KUKA KRL program: ab_st_60301.src, ab_st_60301.dat

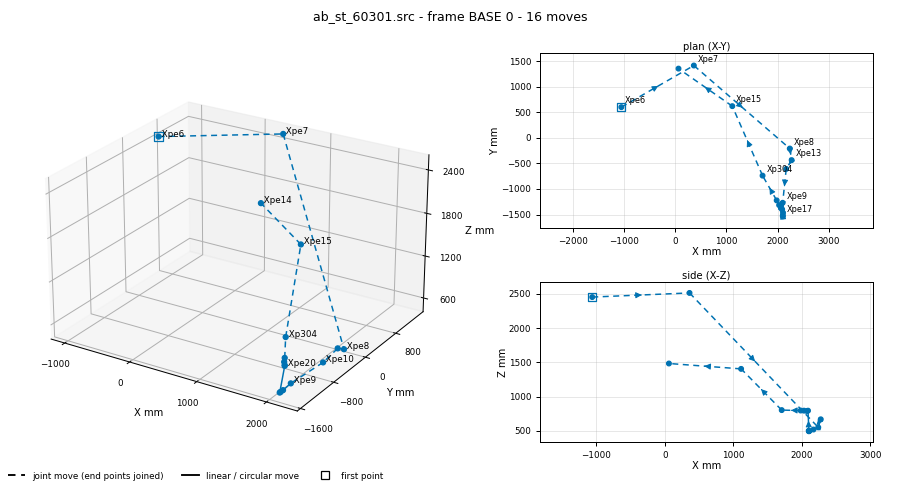
[picture p0: tool path of ab_st_60301.src in frame BASE 0, 16 of 16 moves have a stored position in this frame; points joined in program order, loops and branches not executed]
--- ab_st_60301.src ---
&ACCESS RV2
&REL 437
&COMMENT Deposita Frontal na Geo
&PARAM TEMPLATE = C:\KRC\Roboter\Template\vorgabe
&PARAM EDITMASK = *
DEF ab_st_60301( )
;FOLD INI;%{PE}%V3.2.0,%MKUKATPBASIS,%CINIT,%VCOMMON,%P
;FOLD BAS INI;%{E}%V3.2.0,%MKUKATPBASIS,%CINIT,%VINIT,%P
GLOBAL INTERRUPT DECL 3 WHEN $STOPMESS==TRUE DO IR_STOPM ( )
INTERRUPT ON 3
BAS (#INITMOV,0 )
;ENDFOLD (BAS INI)
;FOLD A20 INI;%{E}%V3.2.0,%MKUKATPA20,%CINIT,%VINIT,%P
IF ARC20==TRUE THEN
A20 (ARC_INI)
INTERRUPT DECL 6 WHEN $CYCFLAG[3]==FALSE DO A20(TECH_STOP2)
ENDIF
;ENDFOLD (A20 INI)
;FOLD A10 INI;%{E}%V3.2.0,%MKUKATPARC,%CINIT,%VINIT,%P
IF A10_OPTION==#ACTIVE THEN
INTERRUPT DECL 4 WHEN $CYCFLAG[2]==FALSE DO A10 (#APPL_ERROR)
INTERRUPT DECL 7 WHEN A_ARC_SWI==#ACTIVE DO A10 (#ARC_SEAM)
INTERRUPT DECL 5 WHEN A_FLY_ARC==TRUE DO A10 (#HPU_ARC)
INTERRUPT  ON 5
A10_INI ( )
ENDIF
;ENDFOLD (A10 INI)
;FOLD GRIPPER INI;%{E}%V3.2.0,%MKUKATPGRIPPER,%CINIT,%VINIT,%P
USER_GRP(0,DUMMY,DUMMY,GDEFAULT)
;ENDFOLD (GRIPPER INI)
;FOLD SPOT INI;%{E}%V3.2.0,%MKUKATPSPOT,%CINIT,%VINIT,%P
USERSPOT(#INIT)
;ENDFOLD (SPOT INI)
;FOLD TOUCHSENSE INI;%{E}%V3.2.0,%MKUKATPTS,%CINIT,%VINIT,%P
IF H70_OPTION THEN
INTERRUPT DECL 15 WHEN $MEAS_PULSE[TOUCH_I[TOUCH_ACTIVE].IN_NR] DO H70 (6,CD0 )
INTERRUPT DECL 16 WHEN $ZERO_MOVE DO H70 (7,CD0 )
INTERRUPT DECL 17 WHEN $TECHPAR_C[FG_TOUCH,8]>0.5 DO H70 (8,CD0)
H70 (1,CD0 )
ENDIF
;ENDFOLD (TOUCHSENSE INI)
;FOLD USER INI;%{E}%V3.2.0,%MKUKATPUSER,%CINIT,%VINIT,%P
;Make your modifications here
;ENDFOLD (USER INI)
;ENDFOLD (INI)

; Caracterização dos meios de produção:
; Versão Atual:
; 19/07/2013 12:00 Name: P13.060-R3 CHANGES: Deposita Frontal Accelo
; na Geobox

chk_w3_wechs_ok ( )        ; ERIFICAÇÃO DE FERRAMENTA: GRIPPER

;FOLD PTP pe6  Vel= 100 % PDAT62 Tool[3]:Gripper Frontal Accelo Base[0];%{PE}%R 4.1.16,%MKUKATPBASIS,%CMOVE,%VPTP,%P 1:PTP, 2:pe6, 3:, 5:100, 7:PDAT62
$BWDSTART = FALSE
PDAT_ACT=PPDAT62
BAS(#PTP_DAT)
FDAT_ACT=Fpe6
BAS(#FRAMES)
BAS(#VEL_PTP,100)
PTP Xpe6
;ENDFOLD

;FOLD WAIT FOR IN 180 'protecao da Garra fechado'  State= TRUE CONT;%{PE}%R 4.1.16,%MKUKATPBASIS,%CWAIT_FOR,%VWAIT_FOR,%P 1:0, 2:180, 3:'protecao da Garra fechado', 5:TRUE, 6:CONTINUE
CONTINUE
WAIT FOR $IN[180]==TRUE
;ENDFOLD

;FOLD PTP pe7 CONT Vel= 65 % PDAT63 Tool[3]:Gripper Frontal Accelo Base[0];%{PE}%R 4.1.16,%MKUKATPBASIS,%CMOVE,%VPTP,%P 1:PTP, 2:pe7, 3:C_PTP, 5:65, 7:PDAT63
$BWDSTART = FALSE
PDAT_ACT=PPDAT63
BAS(#PTP_DAT)
FDAT_ACT=Fpe7
BAS(#FRAMES)
BAS(#VEL_PTP,65)
PTP Xpe7 C_PTP
;ENDFOLD
;FOLD PTP pe8 CONT Vel= 50 % PDAT64 Tool[3]:Gripper Frontal Accelo Base[0];%{PE}%R 4.1.16,%MKUKATPBASIS,%CMOVE,%VPTP,%P 1:PTP, 2:pe8, 3:C_PTP, 5:50, 7:PDAT64
$BWDSTART = FALSE
PDAT_ACT=PPDAT64
BAS(#PTP_DAT)
FDAT_ACT=Fpe8
BAS(#FRAMES)
BAS(#VEL_PTP,50)
PTP Xpe8 C_PTP
;ENDFOLD
;FOLD PTP pe13 CONT Vel= 40 % PDAT69 Tool[3]:Gripper Frontal Accelo Base[0];%{PE}%R 4.1.16,%MKUKATPBASIS,%CMOVE,%VPTP,%P 1:PTP, 2:pe13, 3:C_PTP, 5:40, 7:PDAT69
$BWDSTART = FALSE
PDAT_ACT=PPDAT69
BAS(#PTP_DAT)
FDAT_ACT=Fpe13
BAS(#FRAMES)
BAS(#VEL_PTP,40)
PTP Xpe13 C_PTP
;ENDFOLD
;FOLD PTP pe10 CONT Vel= 40 % PDAT66 Tool[3]:Gripper Frontal Accelo Base[0];%{PE}%R 4.1.16,%MKUKATPBASIS,%CMOVE,%VPTP,%P 1:PTP, 2:pe10, 3:C_PTP, 5:40, 7:PDAT66
$BWDSTART = FALSE
PDAT_ACT=PPDAT66
BAS(#PTP_DAT)
FDAT_ACT=Fpe10
BAS(#FRAMES)
BAS(#VEL_PTP,40)
PTP Xpe10 C_PTP
;ENDFOLD
;FOLD PTP pe9  Vel= 100 % PDAT65 Tool[3]:Gripper Frontal Accelo Base[0];%{PE}%R 4.1.16,%MKUKATPBASIS,%CMOVE,%VPTP,%P 1:PTP, 2:pe9, 3:, 5:100, 7:PDAT65
$BWDSTART = FALSE
PDAT_ACT=PPDAT65
BAS(#PTP_DAT)
FDAT_ACT=Fpe9
BAS(#FRAMES)
BAS(#VEL_PTP,100)
PTP Xpe9
;ENDFOLD

;FOLD OUT 831 'R3 Solic Lib Entregar peca GEOBOX'  State= TRUE CONT;%{PE}%R 4.1.16,%MKUKATPBASIS,%COUT,%VOUTX,%P 2:831, 3:'R3 Solic Lib Entregar peca GEOBOX', 5:TRUE, 6:CONTINUE
CONTINUE
$OUT[831]=TRUE
;ENDFOLD
;FOLD OUT 832 'R3 Entregando peca Geo'  State= TRUE CONT;%{PE}%R 4.1.16,%MKUKATPBASIS,%COUT,%VOUTX,%P 2:832, 3:'R3 Entregando peca Geo', 5:TRUE, 6:CONTINUE
CONTINUE
$OUT[832]=TRUE
;ENDFOLD
;FOLD WAIT FOR IN 832 'Aguarda lib. entrega peca Geo'  State= TRUE ;%{PE}%R 4.1.16,%MKUKATPBASIS,%CWAIT_FOR,%VWAIT_FOR,%P 1:0, 2:832, 3:'Aguarda lib. entrega peca Geo', 5:TRUE, 6:
WAIT FOR $IN[832]==TRUE
;ENDFOLD
;FOLD OUT 832 'R3 Entregando peca Geo'  State= FALSE ;%{PE}%R 4.1.16,%MKUKATPBASIS,%COUT,%VOUTX,%P 2:832, 3:'R3 Entregando peca Geo', 5:FALSE, 6:
$OUT[832]=FALSE
;ENDFOLD
;FOLD OUT 831 'R3 Solic Lib Entregar peca GEOBOX'  State= FALSE ;%{PE}%R 4.1.16,%MKUKATPBASIS,%COUT,%VOUTX,%P 2:831, 3:'R3 Solic Lib Entregar peca GEOBOX', 5:FALSE, 6:
$OUT[831]=FALSE
;ENDFOLD
;FOLD OUT 848 'Area de Solda'  State= FALSE ;%{PE}%R 4.1.16,%MKUKATPBASIS,%COUT,%VOUTX,%P 2:848, 3:'Area de Solda', 5:FALSE, 6:
$OUT[848]=FALSE
;ENDFOLD

;FOLD SET GRP 3  State= OPN  GDAT8;%{PE}%R 4.1.7,%MKUKATPGRP,%CGRP,%VGRP,%P 2:3, 4:1, 5:#NO, 6:GDAT8, 8:0, 10:20
H50(GRP,3,1,GGDAT8)
;ENDFOLD
chk_grp03_opn ( )

;acoplamento geo
;FOLD LIN pbf CONT Vel= 0.3 m/s CPDAT24 Tool[3]:Gripper Frontal Accelo Base[0];%{PE}%R 4.1.16,%MKUKATPBASIS,%CMOVE,%VLIN,%P 1:LIN, 2:pbf, 3:C_DIS, 5:0.3, 7:CPDAT24
$BWDSTART = FALSE
LDAT_ACT=LCPDAT24
BAS(#CP_DAT)
FDAT_ACT=Fpbf
BAS(#FRAMES)
BAS(#VEL_CP,0.3)
LIN Xpbf C_DIS
;ENDFOLD
;FOLD LIN pe17  Vel= 0.2 m/s CPDAT27 Tool[3]:Gripper Frontal Accelo Base[0];%{PE}%R 4.1.16,%MKUKATPBASIS,%CMOVE,%VLIN,%P 1:LIN, 2:pe17, 3:, 5:0.2, 7:CPDAT27
$BWDSTART = FALSE
LDAT_ACT=LCPDAT27
BAS(#CP_DAT)
FDAT_ACT=Fpe17
BAS(#FRAMES)
BAS(#VEL_CP,0.2)
LIN Xpe17
;ENDFOLD

;Posicao de deposito
;FOLD LIN P1000  Vel= 0.1 m/s CPDAT20 Tool[3]:Gripper Frontal Accelo Base[0];%{PE}%R 4.1.16,%MKUKATPBASIS,%CMOVE,%VLIN,%P 1:LIN, 2:P1000, 3:, 5:0.1, 7:CPDAT20
$BWDSTART = FALSE
LDAT_ACT=LCPDAT20
BAS(#CP_DAT)
FDAT_ACT=FP1000
BAS(#FRAMES)
BAS(#VEL_CP,0.1)
LIN XP1000
;ENDFOLD


;FOLD OUT 833 'Solicita lib. sair Geo'  State= TRUE ;%{PE}%R 4.1.16,%MKUKATPBASIS,%COUT,%VOUTX,%P 2:833, 3:'Solicita lib. sair Geo', 5:TRUE, 6:
$OUT[833]=TRUE
;ENDFOLD
;FOLD WAIT FOR IN 834 'aguarda lib. sair Geo'  State= TRUE ;%{PE}%R 4.1.16,%MKUKATPBASIS,%CWAIT_FOR,%VWAIT_FOR,%P 1:0, 2:834, 3:'aguarda lib. sair Geo', 5:TRUE, 6:
WAIT FOR $IN[834]==TRUE
;ENDFOLD
;FOLD OUT 833 'Solicita lib. sair Geo'  State= FALSE ;%{PE}%R 4.1.16,%MKUKATPBASIS,%COUT,%VOUTX,%P 2:833, 3:'Solicita lib. sair Geo', 5:FALSE, 6:
$OUT[833]=FALSE
;ENDFOLD

;FOLD SET GRP 3  State= CLO  GDAT6;%{PE}%R 4.1.7,%MKUKATPGRP,%CGRP,%VGRP,%P 2:3, 4:2, 5:#NO, 6:GDAT6, 8:0, 10:0
H50(GRP,3,2,GGDAT6)
;ENDFOLD
chk_grp03_clo ( )


;FOLD IBUS  OFF;%{PE}%R 4.1.16,%MKUKATPBASIS,%CIBUS,%VMAP,%P 2:#OFF, 3:1
$IBUS_OFF=$IBUS_ON
$IBUS_ON=0
;ENDFOLD
;FOLD WAIT Time= 1.3 sec;%{PE}%R 4.1.16,%MKUKATPBASIS,%CWAIT,%VWAIT,%P 2:1.3
WAIT SEC 1.3
;ENDFOLD
;FOLD OUT 224 'Bloqueio MPS'  State= FALSE ;%{PE}%R 4.1.16,%MKUKATPBASIS,%COUT,%VOUTX,%P 2:224, 3:'Bloqueio MPS', 5:FALSE, 6:
$OUT[224]=FALSE
;ENDFOLD
;FOLD OUT 223 'Desbloqueio MPS'  State= TRUE ;%{PE}%R 4.1.16,%MKUKATPBASIS,%COUT,%VOUTX,%P 2:223, 3:'Desbloqueio MPS', 5:TRUE, 6:
$OUT[223]=TRUE
;ENDFOLD
;FOLD WAIT FOR IN 217 'MPS destravado'  State= TRUE ;%{PE}%R 4.1.16,%MKUKATPBASIS,%CWAIT_FOR,%VWAIT_FOR,%P 1:0, 2:217, 3:'MPS destravado', 5:TRUE, 6:
WAIT FOR $IN[217]==TRUE
;ENDFOLD
;FOLD WAIT FOR IN 221 'MPS travado'  State= FALSE ;%{PE}%R 4.1.16,%MKUKATPBASIS,%CWAIT_FOR,%VWAIT_FOR,%P 1:0, 2:221, 3:'MPS travado', 5:FALSE, 6:
WAIT FOR $IN[221]==FALSE
;ENDFOLD



;FOLD LIN pe20  Vel= 0.2 m/s CPDAT29 Tool[8]:Tool Changer Base[0];%{PE}%R 4.1.16,%MKUKATPBASIS,%CMOVE,%VLIN,%P 1:LIN, 2:pe20, 3:, 5:0.2, 7:CPDAT29
$BWDSTART = FALSE
LDAT_ACT=LCPDAT29
BAS(#CP_DAT)
FDAT_ACT=Fpe20
BAS(#FRAMES)
BAS(#VEL_CP,0.2)
LIN Xpe20
;ENDFOLD
;FOLD LIN pe19  Vel= 0.21 m/s CPDAT30 Tool[8]:Tool Changer Base[0];%{PE}%R 4.1.16,%MKUKATPBASIS,%CMOVE,%VLIN,%P 1:LIN, 2:pe19, 3:, 5:0.21, 7:CPDAT30
$BWDSTART = FALSE
LDAT_ACT=LCPDAT30
BAS(#CP_DAT)
FDAT_ACT=Fpe19
BAS(#FRAMES)
BAS(#VEL_CP,0.21)
LIN Xpe19
;ENDFOLD




;FOLD LIN P1001 CONT Vel= 0.1 m/s CPDAT21 Tool[8]:Tool Changer Base[0];%{PE}%R 4.1.16,%MKUKATPBASIS,%CMOVE,%VLIN,%P 1:LIN, 2:P1001, 3:C_DIS, 5:0.1, 7:CPDAT21
$BWDSTART = FALSE
LDAT_ACT=LCPDAT21
BAS(#CP_DAT)
FDAT_ACT=FP1001
BAS(#FRAMES)
BAS(#VEL_CP,0.1)
LIN XP1001 C_DIS
;ENDFOLD

;FOLD OUT 848 'Area de Solda'  State= TRUE ;%{PE}%R 4.1.16,%MKUKATPBASIS,%COUT,%VOUTX,%P 2:848, 3:'Area de Solda', 5:TRUE, 6:
$OUT[848]=TRUE
;ENDFOLD
;FOLD PULSE 847 'Peca na Geo'  State= TRUE   Time= 3 sec;%{PE}%R 4.1.16,%MKUKATPBASIS,%COUT,%VPULSE,%P 2:847, 3:'Peca na Geo', 5:TRUE, 6:, 8:3
PULSE($OUT[847], TRUE,3)
;ENDFOLD

;FOLD LIN p303 CONT Vel= 0.8 m/s CPDAT13 Tool[8]:Tool Changer Base[0];%{PE}%R 4.1.16,%MKUKATPBASIS,%CMOVE,%VLIN,%P 1:LIN, 2:p303, 3:C_DIS, 5:0.8, 7:CPDAT13
$BWDSTART = FALSE
LDAT_ACT=LCPDAT13
BAS(#CP_DAT)
FDAT_ACT=Fp303
BAS(#FRAMES)
BAS(#VEL_CP,0.8)
LIN Xp303 C_DIS
;ENDFOLD

;FOLD PTP p304 CONT Vel= 100 % PDAT47 Tool[8]:Tool Changer Base[0];%{PE}%R 4.1.16,%MKUKATPBASIS,%CMOVE,%VPTP,%P 1:PTP, 2:p304, 3:C_PTP, 5:100, 7:PDAT47
$BWDSTART = FALSE
PDAT_ACT=PPDAT47
BAS(#PTP_DAT)
FDAT_ACT=Fp304
BAS(#FRAMES)
BAS(#VEL_PTP,100)
PTP Xp304 C_PTP
;ENDFOLD

;FOLD OUT 223 'Desbloqueio MPS'  State= FALSE CONT;%{PE}%R 4.1.16,%MKUKATPBASIS,%COUT,%VOUTX,%P 2:223, 3:'Desbloqueio MPS', 5:FALSE, 6:CONTINUE
CONTINUE
$OUT[223]=FALSE
;ENDFOLD
;FOLD OUT 832 'R3 Entregando peca Geo'  State= TRUE CONT;%{PE}%R 4.1.16,%MKUKATPBASIS,%COUT,%VOUTX,%P 2:832, 3:'R3 Entregando peca Geo', 5:TRUE, 6:CONTINUE
CONTINUE
$OUT[832]=TRUE
;ENDFOLD

;FOLD Kollision.Ueberwachung_4_Aus ;%{PE}%MKUKATPUSER
COLLSTOP( 4, 2 )
;ENDFOLD

;FOLD PULSE 834 'Entregou peca Geo'  State= TRUE   Time= 3 sec;%{PE}%R 4.1.16,%MKUKATPBASIS,%COUT,%VPULSE,%P 2:834, 3:'Entregou peca Geo', 5:TRUE, 6:, 8:3
PULSE($OUT[834], TRUE,3)
;ENDFOLD
;FOLD PULSE 175 'Proteção da pinca C1 abrir'  State= TRUE   Time= 3 sec;%{PE}%R 4.1.16,%MKUKATPBASIS,%COUT,%VPULSE,%P 2:175, 3:'Proteção da pinca C1 abrir', 5:TRUE, 6:, 8:3
PULSE($OUT[175], TRUE,3)
;ENDFOLD

;FOLD PTP pe15 CONT Vel= 100 % PDAT71 Tool[8]:Tool Changer Base[0];%{PE}%R 4.1.16,%MKUKATPBASIS,%CMOVE,%VPTP,%P 1:PTP, 2:pe15, 3:C_PTP, 5:100, 7:PDAT71
$BWDSTART = FALSE
PDAT_ACT=PPDAT71
BAS(#PTP_DAT)
FDAT_ACT=Fpe15
BAS(#FRAMES)
BAS(#VEL_PTP,100)
PTP Xpe15 C_PTP
;ENDFOLD
;FOLD PTP pe14  Vel= 100 % PDAT70 Tool[8]:Tool Changer Base[0];%{PE}%R 4.1.16,%MKUKATPBASIS,%CMOVE,%VPTP,%P 1:PTP, 2:pe14, 3:, 5:100, 7:PDAT70
$BWDSTART = FALSE
PDAT_ACT=PPDAT70
BAS(#PTP_DAT)
FDAT_ACT=Fpe14
BAS(#FRAMES)
BAS(#VEL_PTP,100)
PTP Xpe14
;ENDFOLD

END

--- ab_st_60301.dat ---
&ACCESS RV2
&REL 437
&COMMENT Deposita Frontal na Geo
&PARAM TEMPLATE = C:\KRC\Roboter\Template\vorgabe
&PARAM EDITMASK = *
DEFDAT  AB_ST_60301
;FOLD EXTERNAL DECLARATIONS;%{PE}%V3.2.0,%MKUKATPBASIS,%CEXT,%VCOMMON,%P
;FOLD BAS EXT;%{PE}%V3.2.0,%MKUKATPBASIS,%CEXT,%VEXT,%P
EXT  BAS (BAS_COMMAND  :IN,REAL  :IN )
DECL INT SUCCESS
;ENDFOLD
;FOLD A10 EXT;%{E}%V3.2.0,%MKUKATPARC,%CEXT,%VEXT,%P
EXT  A10 (A_CMD_T  :IN,A_STRT_T  :IN,A_WELD_T  :IN,A_END_T  :IN,INT  :IN )
;ENDFOLD
;FOLD A20 EXT;%{E}%V3.2.0,%MKUKATPA20,%CEXT,%VEXT,%P
EXT  A20 (INT  :IN,WELD_ST  :IN,WELD_FI  :IN,INT  :IN )
;ENDFOLD
;FOLD GRIPPER EXT;%{E}%V3.2.0,%MKUKATPGRIPPER,%CEXT,%VEXT,%P
EXT  H50 (INT  :IN,INT  :IN,INT  :IN,GRP_TYP  :IN )
;ENDFOLD
;FOLD SPOT EXT;%{E}%V3.2.0,%MKUKATPSPOT,%CEXT,%VEXT,%P
EXT  USERSPOT (S_COMMAND  :IN,SPOT_TYPE  :IN )
;ENDFOLD
;FOLD TOUCHSENSE EXT;%{E}%V3.2.0,%MKUKATPTS,%CEXT,%VEXT,%P
EXT  H70 (INT  :IN,SRCH_TYP_2  :OUT,E6POS  :IN,SRCH_TYP_3  :IN,SRCH_TYP_2  :IN,SRCH_TYP_2  :IN,SRCH_TYP_2  :IN,SRCH_TYP_2  :IN,SRCH_TYP_2  :IN,INT  :IN )
;ENDFOLD
;FOLD USER EXT;%{E}%V3.2.0,%MKUKATPUSER,%CEXT,%VEXT,%P
;Make here your modifications
;ENDFOLD
;ENDFOLD

DECL BASIS_SUGG_T LAST_BASIS={POINT1[] "pe24                    ",POINT2[] "pe24                    ",CP_PARAMS[] "CPDAT28                 ",PTP_PARAMS[] "PDAT77                  ",CONT[] "                        ",CP_VEL[] "0.1                     ",PTP_VEL[] "40                      "}
DECL E6POS XP1={x -188.3992,y 2368.7981,z 816.157471,a 0.682591379,b 56.9728508,c -155.483307,s 6,t 51,e1 0.0,e2 0.0,e3 0.0,e4 0.0,e5 0.0,e6 0.0}


DECL FDAT FP1={TOOL_NO 8,BASE_NO 0,IPO_FRAME #BASE}
DECL PDAT PPDAT1={VEL 100.0,ACC 100.0,APO_DIST 100.0}
DECL E6POS XP2={x 39.6335411,y 2248.2561,z 963.446594,a 0.683832824,b 56.9725304,c -155.481995,s 6,t 51,e1 0.0,e2 0.0,e3 0.0,e4 0.0,e5 0.0,e6 0.0}
DECL FDAT FP2={TOOL_NO 8,BASE_NO 0,IPO_FRAME #BASE}
DECL PDAT PPDAT2={VEL 100.0,ACC 100.0,APO_DIST 100.0}
DECL E6POS XP3={x 388.941711,y 1754.29297,z 2068.00708,a 129.908005,b 79.1631622,c 52.0251884,s 2,t 35,e1 0.0,e2 0.0,e3 0.0,e4 0.0,e5 0.0,e6 0.0}
DECL FDAT FP3={TOOL_NO 8,BASE_NO 0,IPO_FRAME #BASE}
DECL PDAT PPDAT3={VEL 100.0,ACC 100.0,APO_DIST 100.0}
DECL E6POS XP4={x -141.421799,y 2321.63794,z 903.706726,a -12.8919296,b 56.8668289,c -155.093994,s 6,t 51,e1 0.0,e2 0.0,e3 0.0,e4 0.0,e5 0.0,e6 0.0}

DECL FDAT FP4={TOOL_NO 8,BASE_NO 0,IPO_FRAME #BASE}
DECL PDAT PPDAT4={VEL 100.0,ACC 100.0,APO_DIST 100.0}
DECL E6POS XP5={x -310.951813,y 2507.78101,z 762.400391,a -5.76357794,b 56.6388206,c -155.210098,s 6,t 51,e1 0.0,e2 0.0,e3 0.0,e4 0.0,e5 0.0,e6 0.0}
DECL FDAT FP5={TOOL_NO 8,BASE_NO 0,IPO_FRAME #BASE}
DECL PDAT PPDAT5={VEL 100.0,ACC 100.0,APO_DIST 100.0}
DECL E6POS XP6={x -231.908905,y 2732.73511,z 874.473572,a 62.2883606,b -0.0793622211,c -89.9837265,s 6,t 51,e1 0.0,e2 0.0,e3 0.0,e4 0.0,e5 0.0,e6 0.0}
DECL FDAT FP6={TOOL_NO 3,BASE_NO 0,IPO_FRAME #BASE}
DECL PDAT PPDAT6={VEL 100.0,ACC 100.0,APO_DIST 100.0}
DECL E6POS XP7={x -138.7957,y 2749.80103,z 865.714417,a 64.2388,b -0.0770005435,c -89.9825897,s 6,t 51,e1 0.0,e2 0.0,e3 0.0,e4 0.0,e5 0.0,e6 0.0}
DECL FDAT FP7={TOOL_NO 3,BASE_NO 0,IPO_FRAME #BASE}
DECL PDAT PPDAT7={VEL 100.0,ACC 100.0,APO_DIST 100.0}
DECL E6POS XP8={x -58.7346306,y 2732.94092,z 865.675293,a 67.7668915,b -0.075337939,c -89.9879227,s 6,t 51,e1 0.0,e2 0.0,e3 0.0,e4 0.0,e5 0.0,e6 0.0}
DECL FDAT FP8={TOOL_NO 3,BASE_NO 0,IPO_FRAME #BASE}
DECL PDAT PPDAT8={VEL 100.0,ACC 100.0,APO_DIST 100.0}
DECL E6POS XP9={x -4.80422878,y 2723.65308,z 865.806519,a 69.4628601,b -0.0796707496,c -89.9865265,s 6,t 51,e1 0.0,e2 0.0,e3 0.0,e4 0.0,e5 0.0,e6 0.0}
DECL FDAT FP9={TOOL_NO 3,BASE_NO 0,IPO_FRAME #BASE}
DECL PDAT PPDAT9={VEL 100.0,ACC 100.0,APO_DIST 100.0}
DECL E6POS XP10={x 96.421463,y 2705.94312,z 852.752686,a 59.7485199,b -0.0976489186,c -89.969368,s 6,t 51,e1 0.0,e2 0.0,e3 0.0,e4 0.0,e5 0.0,e6 0.0}
DECL FDAT FP10={TOOL_NO 3,BASE_NO 0,IPO_FRAME #BASE}
DECL PDAT PPDAT10={VEL 100.0,ACC 100.0,APO_DIST 100.0}
DECL E6POS XP11={x 254.399094,y 2660.85889,z 851.276611,a 47.4197311,b -0.094424963,c -89.9508286,s 6,t 51,e1 0.0,e2 0.0,e3 0.0,e4 0.0,e5 0.0,e6 0.0}
DECL FDAT FP11={TOOL_NO 3,BASE_NO 0,IPO_FRAME #BASE}
DECL PDAT PPDAT11={VEL 100.0,ACC 100.0,APO_DIST 100.0}
DECL E6POS XP12={x 254.197098,y 2660.07202,z 1289.99695,a 47.4186096,b -0.0936179385,c -90.4839935,s 6,t 51,e1 0.0,e2 0.0,e3 0.0,e4 0.0,e5 0.0,e6 0.0}
DECL FDAT FP12={TOOL_NO 3,BASE_NO 0,IPO_FRAME #BASE}
DECL PDAT PPDAT12={VEL 100.0,ACC 100.0,APO_DIST 100.0}
DECL E6POS XP13={x 387.00351,y 2537.04199,z 1725.88306,a 47.4178085,b -0.0868179128,c -81.4952316,s 6,t 51,e1 0.0,e2 0.0,e3 0.0,e4 0.0,e5 0.0,e6 0.0}
DECL FDAT FP13={TOOL_NO 3,BASE_NO 0,IPO_FRAME #BASE}
DECL PDAT PPDAT13={VEL 100.0,ACC 100.0,APO_DIST 100.0}
DECL E6POS XP14={x 577.404114,y 2286.39795,z 1935.52197,a 30.7294006,b 4.42975616,c -75.2716522,s 6,t 51,e1 0.0,e2 0.0,e3 0.0,e4 0.0,e5 0.0,e6 0.0}
DECL FDAT FP14={TOOL_NO 3,BASE_NO 0,IPO_FRAME #BASE}
DECL PDAT PPDAT14={VEL 100.0,ACC 100.0,APO_DIST 100.0}
DECL E6POS XP15={x -210.601395,y 2793.87988,z 858.125427,a 47.6891098,b -0.311072499,c -90.0127563,s 6,t 51,e1 0.0,e2 0.0,e3 0.0,e4 0.0,e5 0.0,e6 0.0}
DECL FDAT FP15={TOOL_NO 3,BASE_NO 0,IPO_FRAME #BASE}
DECL PDAT PPDAT15={VEL 100.0,ACC 100.0,APO_DIST 100.0}
DECL LDAT LCPDAT1={VEL 2.0,ACC 100.0,APO_DIST 100.0,APO_FAC 50.0}
DECL E6POS XP16={x -253.589203,y 2420.03198,z 826.688293,a -15.0486002,b 56.5221214,c -156.482697,s 6,t 51,e1 0.0,e2 0.0,e3 0.0,e4 0.0,e5 0.0,e6 0.0}
DECL FDAT FP16={TOOL_NO 8,BASE_NO 0,IPO_FRAME #BASE}
DECL LDAT LCPDAT2={VEL 2.0,ACC 100.0,APO_DIST 100.0,APO_FAC 50.0}
DECL LDAT LCPDAT3={VEL 2.0,ACC 100.0,APO_DIST 100.0,APO_FAC 50.0}
DECL E6POS XP17={x -104.003502,y 2593.61499,z 862.898682,a 47.8507004,b -0.443317294,c -89.9662323,s 6,t 51,e1 0.0,e2 0.0,e3 0.0,e4 0.0,e5 0.0,e6 0.0}
DECL FDAT FP17={TOOL_NO 3,BASE_NO 0,IPO_FRAME #BASE}
DECL PDAT PPDAT16={VEL 100.0,ACC 100.0,APO_DIST 100.0}
DECL E6POS XP18={x -114.378899,y 2558.99609,z 1228.50195,a 42.74683,b -0.281747609,c -89.6939468,s 6,t 51,e1 0.0,e2 0.0,e3 0.0,e4 0.0,e5 0.0,e6 0.0}
DECL FDAT FP18={TOOL_NO 3,BASE_NO 0,IPO_FRAME #BASE}
DECL PDAT PPDAT17={VEL 100.0,ACC 100.0,APO_DIST 100.0}
DECL E6POS XP19={x 59.8382301,y 2366.573,z 1678.95105,a 32.0545197,b 2.27294707,c -77.4810028,s 6,t 51,e1 0.0,e2 0.0,e3 0.0,e4 0.0,e5 0.0,e6 0.0}
DECL FDAT FP19={TOOL_NO 3,BASE_NO 0,IPO_FRAME #BASE}
DECL PDAT PPDAT18={VEL 100.0,ACC 100.0,APO_DIST 100.0}
DECL E6POS XP20={x 178.339905,y 2018.22302,z 1695.13098,a 16.4725895,b 3.63115811,c -69.0822067,s 6,t 51,e1 0.0,e2 0.0,e3 0.0,e4 0.0,e5 0.0,e6 0.0}
DECL FDAT FP20={TOOL_NO 3,BASE_NO 0,IPO_FRAME #BASE}
DECL PDAT PPDAT19={VEL 100.0,ACC 100.0,APO_DIST 100.0}
DECL E6POS XP21={x 103.363403,y 1772.48596,z 1818.14697,a 12.0467701,b 4.32170582,c -60.2828217,s 6,t 51,e1 0.0,e2 0.0,e3 0.0,e4 0.0,e5 0.0,e6 0.0}
DECL FDAT FP21={TOOL_NO 3,BASE_NO 0,IPO_FRAME #BASE}
DECL PDAT PPDAT20={VEL 100.0,ACC 100.0,APO_DIST 100.0}
DECL E6POS XP22={x 2104.2251,y 68.1197662,z 102.1996,a -0.666801214,b -0.144442394,c -152.486694,s 2,t 3,e1 0.0,e2 0.0,e3 0.0,e4 0.0,e5 0.0,e6 0.0}
DECL FDAT FP22={TOOL_NO 3,BASE_NO 0,IPO_FRAME #BASE}
DECL PDAT PPDAT21={VEL 100.0,ACC 100.0,APO_DIST 100.0}
DECL E6POS XP23={x -1056.99194,y 600.572815,z 2451.80591,a 175.843597,b -72.5620575,c 179.205307,s 2,t 3,e1 0.0,e2 0.0,e3 0.0,e4 0.0,e5 0.0,e6 0.0}
DECL FDAT FP23={TOOL_NO 3,BASE_NO 0,IPO_FRAME #BASE}
DECL PDAT PPDAT22={VEL 100.0,ACC 100.0,APO_DIST 100.0}
DECL E6POS XP24={x -1468.95703,y 1158.19897,z 2120.92505,a 177.713699,b -54.6900291,c 178.097107,s 2,t 11,e1 0.0,e2 0.0,e3 0.0,e4 0.0,e5 0.0,e6 0.0}
DECL FDAT FP24={TOOL_NO 3,BASE_NO 0,IPO_FRAME #BASE}
DECL PDAT PPDAT23={VEL 100.0,ACC 100.0,APO_DIST 100.0}
DECL E6POS XP25={x -1983.53406,y 1198.328,z 537.303406,a 179.117096,b 7.47287893,c -179.832199,s 2,t 3,e1 0.0,e2 0.0,e3 0.0,e4 0.0,e5 0.0,e6 0.0}
DECL FDAT FP25={TOOL_NO 3,BASE_NO 0,IPO_FRAME #BASE}
DECL PDAT PPDAT24={VEL 100.0,ACC 100.0,APO_DIST 100.0}
DECL E6POS XP26={x -1884.86902,y 1143.23401,z -12.8902597,a 178.553894,b 27.9167995,c -179.580795,s 2,t 3,e1 0.0,e2 0.0,e3 0.0,e4 0.0,e5 0.0,e6 0.0}
DECL FDAT FP26={TOOL_NO 3,BASE_NO 0,IPO_FRAME #BASE}
DECL PDAT PPDAT25={VEL 100.0,ACC 100.0,APO_DIST 100.0}
DECL E6POS XP27={x -1983.52502,y 1198.323,z 537.230286,a 179.116501,b 7.47453594,c -179.831207,s 2,t 3,e1 0.0,e2 0.0,e3 0.0,e4 0.0,e5 0.0,e6 0.0}
DECL FDAT FP27={TOOL_NO 3,BASE_NO 0,IPO_FRAME #BASE}
DECL PDAT PPDAT26={VEL 100.0,ACC 100.0,APO_DIST 100.0}
DECL E6POS XP28={x -1795.58105,y 1198.05896,z 1268.58801,a 179.125305,b -28.5398693,c -179.794601,s 2,t 3,e1 0.0,e2 0.0,e3 0.0,e4 0.0,e5 0.0,e6 0.0}
DECL FDAT FP28={TOOL_NO 3,BASE_NO 0,IPO_FRAME #BASE}
DECL PDAT PPDAT27={VEL 100.0,ACC 100.0,APO_DIST 100.0}
DECL E6POS XP29={x -1468.95703,y 1158.19397,z 2120.92896,a 177.714005,b -54.690239,c 178.096802,s 2,t 11,e1 0.0,e2 0.0,e3 0.0,e4 0.0,e5 0.0,e6 0.0}
DECL FDAT FP29={TOOL_NO 3,BASE_NO 0,IPO_FRAME #BASE}
DECL PDAT PPDAT28={VEL 100.0,ACC 100.0,APO_DIST 100.0}
DECL E6POS XP30={x 103.363403,y 1772.48596,z 1818.14697,a 12.0467701,b 4.32170582,c -60.2828217,s 6,t 51,e1 0.0,e2 0.0,e3 0.0,e4 0.0,e5 0.0,e6 0.0}
DECL FDAT FP30={TOOL_NO 3,BASE_NO 0,IPO_FRAME #BASE}
DECL PDAT PPDAT29={VEL 100.0,ACC 100.0,APO_DIST 100.0}
DECL E6POS XP31={x 178.339905,y 2018.22302,z 1695.13098,a 16.4725895,b 3.63115811,c -69.0822067,s 6,t 51,e1 0.0,e2 0.0,e3 0.0,e4 0.0,e5 0.0,e6 0.0}
DECL FDAT FP31={TOOL_NO 3,BASE_NO 0,IPO_FRAME #BASE}
DECL PDAT PPDAT30={VEL 100.0,ACC 100.0,APO_DIST 100.0}
DECL E6POS XP32={x 59.8382301,y 2366.573,z 1678.95105,a 32.0545197,b 2.27294707,c -77.4810028,s 6,t 51,e1 0.0,e2 0.0,e3 0.0,e4 0.0,e5 0.0,e6 0.0}
DECL FDAT FP32={TOOL_NO 3,BASE_NO 0,IPO_FRAME #BASE}
DECL PDAT PPDAT31={VEL 100.0,ACC 100.0,APO_DIST 100.0}
DECL E6POS XP33={x -114.378899,y 2558.99609,z 1228.50195,a 42.74683,b -0.281747609,c -89.6939468,s 6,t 51,e1 0.0,e2 0.0,e3 0.0,e4 0.0,e5 0.0,e6 0.0}
DECL FDAT FP33={TOOL_NO 3,BASE_NO 0,IPO_FRAME #BASE}
DECL PDAT PPDAT32={VEL 100.0,ACC 100.0,APO_DIST 100.0}
DECL E6POS XP34={x -69.7102814,y 2637.021,z 863.732788,a 46.0948906,b -0.300397307,c -89.7107086,s 6,t 51,e1 0.0,e2 0.0,e3 0.0,e4 0.0,e5 0.0,e6 0.0}
DECL FDAT FP34={TOOL_NO 3,BASE_NO 0,IPO_FRAME #BASE}
DECL PDAT PPDAT33={VEL 100.0,ACC 100.0,APO_DIST 100.0}
DECL E6POS XP35={x -217.495407,y 2798.87402,z 862.13623,a 47.7863503,b -0.181169301,c -89.6277924,s 6,t 51,e1 0.0,e2 0.0,e3 0.0,e4 0.0,e5 0.0,e6 0.0}
DECL FDAT FP35={TOOL_NO 3,BASE_NO 0,IPO_FRAME #BASE}
DECL PDAT PPDAT34={VEL 100.0,ACC 100.0,APO_DIST 100.0}
DECL E6POS XP36={x -217.537292,y 2799.2251,z 752.995728,a 48.2843094,b -0.3213332,c -89.7200928,s 6,t 51,e1 0.0,e2 0.0,e3 0.0,e4 0.0,e5 0.0,e6 0.0}
DECL FDAT FP36={TOOL_NO 3,BASE_NO 0,IPO_FRAME #BASE}
DECL LDAT LCPDAT4={VEL 2.0,ACC 100.0,APO_DIST 100.0,APO_FAC 50.0}
DECL E6POS XP37={x -218.973099,y 2799.72998,z 833.772522,a 48.4467506,b -0.344602793,c -89.9268036,s 6,t 51,e1 0.0,e2 0.0,e3 0.0,e4 0.0,e5 0.0,e6 0.0}
DECL FDAT FP37={TOOL_NO 3,BASE_NO 0,IPO_FRAME #BASE}
DECL LDAT LCPDAT5={VEL 2.0,ACC 100.0,APO_DIST 100.0,APO_FAC 50.0}
DECL E6POS XP38={x -334.715088,y 2494.78711,z 762.013611,a -15.0434103,b 56.5220718,c -156.471695,s 6,t 51,e1 0.0,e2 0.0,e3 0.0,e4 0.0,e5 0.0,e6 0.0}
DECL FDAT FP38={TOOL_NO 8,BASE_NO 0,IPO_FRAME #BASE}
DECL LDAT LCPDAT6={VEL 2.0,ACC 100.0,APO_DIST 100.0,APO_FAC 50.0}
DECL E6POS XP39={x -2416.61401,y 39.1588516,z 1046.82495,a -174.215302,b -7.00384188,c 141.212906,s 2,t 3,e1 0.0,e2 0.0,e3 0.0,e4 0.0,e5 0.0,e6 0.0}
DECL FDAT FP39={TOOL_NO 3,BASE_NO 2,IPO_FRAME #BASE}
DECL PDAT PPDAT35={VEL 100.0,ACC 60.0,APO_DIST 30.0}
DECL E6POS XP40={x 2290.56299,y -695.490601,z 1091.52795,a 74.2140274,b 81.0776062,c 153.915894,s 2,t 2,e1 0.0,e2 0.0,e3 0.0,e4 0.0,e5 0.0,e6 0.0}
DECL FDAT FP40={TOOL_NO 3,BASE_NO 0,IPO_FRAME #BASE}
DECL PDAT PPDAT36={VEL 100.0,ACC 100.0,APO_DIST 100.0}
DECL E6POS XP41={x 2120.95801,y -1006.67102,z 519.729919,a 146.695801,b 89.4882584,c -122.776802,s 2,t 2,e1 0.0,e2 0.0,e3 0.0,e4 0.0,e5 0.0,e6 0.0}
DECL FDAT FP41={TOOL_NO 3,BASE_NO 0,IPO_FRAME #BASE}
DECL PDAT PPDAT37={VEL 100.0,ACC 100.0,APO_DIST 100.0}
DECL E6POS XP42={x 2103.9519,y -1494.86694,z 502.313507,a -90.9648972,b 89.7392731,c -0.781405687,s 2,t 2,e1 0.0,e2 0.0,e3 0.0,e4 0.0,e5 0.0,e6 0.0}
DECL FDAT FP42={TOOL_NO 3,BASE_NO 0,IPO_FRAME #BASE}
DECL PDAT PPDAT38={VEL 100.0,ACC 100.0,APO_DIST 100.0}
DECL E6POS XP43={x 2100.85596,y -1376.36096,z 502.189606,a 172.303299,b 89.4688568,c -98.2193222,s 2,t 2,e1 0.0,e2 0.0,e3 0.0,e4 0.0,e5 0.0,e6 0.0}
DECL FDAT FP43={TOOL_NO 3,BASE_NO 0,IPO_FRAME #BASE}
DECL LDAT LCPDAT7={VEL 2.0,ACC 85.0,APO_DIST 10.0,APO_FAC 50.0}
DECL E6POS XP44={x 2105.36499,y -1049.36401,z 552.007874,a -90.6014099,b 89.7380829,c -0.414461106,s 2,t 2,e1 0.0,e2 0.0,e3 0.0,e4 0.0,e5 0.0,e6 0.0}
DECL FDAT FP44={TOOL_NO 3,BASE_NO 0,IPO_FRAME #BASE}
DECL PDAT PPDAT39={VEL 100.0,ACC 100.0,APO_DIST 100.0}
DECL E6POS XTESTE={x -218.994202,y 2799.72998,z 855.550476,a 48.4468689,b -0.344231814,c -89.9264526,s 6,t 51,e1 0.0,e2 0.0,e3 0.0,e4 0.0,e5 0.0,e6 0.0}
DECL FDAT Fteste={TOOL_NO 3,BASE_NO 0,IPO_FRAME #BASE}
DECL LDAT LCPDAT8={VEL 2.0,ACC 100.0,APO_DIST 100.0,APO_FAC 50.0}
DECL E6POS XP200={x -318.375702,y 2479.64697,z 775.077576,a -15.0468197,b 56.522541,c -156.479507,s 6,t 51,e1 0.0,e2 0.0,e3 0.0,e4 0.0,e5 0.0,e6 0.0}
DECL FDAT Fp200={TOOL_NO 8,BASE_NO 0,IPO_FRAME #BASE}
DECL LDAT LCPDAT9={VEL 2.0,ACC 100.0,APO_DIST 100.0,APO_FAC 50.0}
DECL PDAT PPDAT40={VEL 100.0,ACC 100.0,APO_DIST 100.0}
DECL E6POS XP60={x -1795.57996,y 1198.06104,z 1268.58301,a 179.124603,b -28.5397491,c -179.794098,s 2,t 3,e1 0.0,e2 0.0,e3 0.0,e4 0.0,e5 0.0,e6 0.0}
DECL FDAT Fp60={TOOL_NO 3,BASE_NO 0,IPO_FRAME #BASE}
DECL PDAT PPDAT41={VEL 100.0,ACC 100.0,APO_DIST 100.0}
DECL E6POS XP61={x -1883.59094,y 1144.84204,z -110.182701,a 178.551804,b 28.0140095,c -179.494507,s 2,t 3,e1 0.0,e2 0.0,e3 0.0,e4 0.0,e5 0.0,e6 0.0}
DECL FDAT Fp61={TOOL_NO 3,BASE_NO 0,IPO_FRAME #BASE}
DECL LDAT LCPDAT10={VEL 2.0,ACC 100.0,APO_DIST 100.0,APO_FAC 50.0}
DECL GRP_SUGG_T LAST_GRP={NUMBER[] "3                       ",STATE[] "1                       ",PARAMS[] "GDAT8                   "}
DECL GRP_TYP GCONT={G_APO #YES,TIME 0.0,CTRL #OFF,DLY 0,DST 0}
DECL GRP_TYP GGDAT0={G_APO #NO,TIME 0.200000003,CTRL #OFF,DLY 0,DST 1}
DECL GRP_TYP GGDAT1={G_APO #NO,TIME 0.200000003,CTRL #OFF,DLY 0,DST 1}
DECL GRP_TYP GGDAT2={G_APO #NO,TIME 0.200000003,CTRL #OFF,DLY 0,DST 1}
DECL GRP_TYP GGDAT3={G_APO #NO,TIME 0.200000003,CTRL #OFF,DLY 0,DST 1}
DECL GRP_TYP GGDAT4={G_APO #NO,TIME 0.200000003,CTRL #OFF,DLY 0,DST 1}
DECL FDAT FHOME1={TOOL_NO 3,BASE_NO 0,IPO_FRAME #BASE}
DECL E6POS XP62={x -2045.90601,y 1149.81104,z 208.532593,a 178.554001,b 27.91716,c -179.580902,s 2,t 3,e1 0.0,e2 0.0,e3 0.0,e4 0.0,e5 0.0,e6 0.0}
DECL FDAT Fp62={TOOL_NO 3,BASE_NO 0,IPO_FRAME #BASE}
DECL LDAT LCPDAT11={VEL 2.0,ACC 100.0,APO_DIST 100.0,APO_FAC 50.0}
DECL PDAT PPDAT42={VEL 100.0,ACC 100.0,APO_DIST 100.0}
DECL PDAT PPDAT43={VEL 100.0,ACC 75.0,APO_DIST 100.0}
DECL FDAT FHOME2={TOOL_NO 3,BASE_NO 0,IPO_FRAME #BASE}
DECL PDAT PPDAT44={VEL 100.0,ACC 80.0,APO_DIST 20.0}
DECL GRP_TYP GGDAT5={G_APO #NO,TIME 0.200000003,CTRL #OFF,DLY 0,DST 1}
DECL GRP_TYP GGDAT6={G_APO #NO,TIME 0.5,CTRL #OFF,DLY 0,DST 1}
DECL E6POS XP300={x 2103.87793,y -1542.31702,z 502.337585,a -91.9767227,b 89.7423706,c -1.79670501,s 2,t 2,e1 0.0,e2 0.0,e3 0.0,e4 0.0,e5 0.0,e6 0.0}
DECL FDAT Fp300={TOOL_NO 3,BASE_NO 0,IPO_FRAME #BASE}
DECL PDAT PPDAT45={VEL 100.0,ACC 100.0,APO_DIST 100.0}
DECL E6POS XP301={x 2101.01196,y -1428.62,z 807.025513,a 29.7582302,b 15.1351204,c 89.7658234,s 2,t 2,e1 0.0,e2 0.0,e3 0.0,e4 0.0,e5 0.0,e6 0.0}
DECL FDAT Fp301={TOOL_NO 8,BASE_NO 0,IPO_FRAME #BASE}
DECL PDAT PPDAT46={VEL 100.0,ACC 100.0,APO_DIST 100.0}
DECL E6POS XP302={x 1998.20703,y -1249.63599,z 806.080017,a 29.7583504,b 15.1435204,c 89.7742615,s 2,t 2,e1 0.0,e2 0.0,e3 0.0,e4 0.0,e5 0.0,e6 0.0}
DECL FDAT Fp302={TOOL_NO 8,BASE_NO 0,IPO_FRAME #BASE}
DECL LDAT LCPDAT12={VEL 2.0,ACC 100.0,APO_DIST 100.0,APO_FAC 50.0}
DECL E6POS XP303={x 1982.17505,y -1223.79004,z 797.602417,a 29.8996201,b 15.00529,c 89.9983521,s 2,t 2,e1 0.0,e2 0.0,e3 0.0,e4 0.0,e5 0.0,e6 0.0}
DECL FDAT Fp303={TOOL_NO 8,BASE_NO 0,IPO_FRAME #BASE}
DECL LDAT LCPDAT13={VEL 2.0,ACC 85.0,APO_DIST 20.0,APO_FAC 50.0}
DECL E6POS XP304={x 1705.78699,y -739.28833,z 803.88092,a 29.7551403,b 15.1431599,c 89.7668915,s 2,t 2,e1 0.0,e2 0.0,e3 0.0,e4 0.0,e5 0.0,e6 0.0}
DECL FDAT Fp304={TOOL_NO 8,BASE_NO 0,IPO_FRAME #BASE}
DECL PDAT PPDAT47={VEL 100.0,ACC 100.0,APO_DIST 50.0}
DECL E6POS XP305={x -215.8284,y 2796.93311,z 843.476013,a 47.9605103,b 0.0409639515,c -90.3939896,s 6,t 51,e1 0.0,e2 0.0,e3 0.0,e4 0.0,e5 0.0,e6 0.0}
DECL FDAT Fp305={TOOL_NO 3,BASE_NO 0,IPO_FRAME #BASE}
DECL LDAT LCPDAT15={VEL 2.0,ACC 100.0,APO_DIST 100.0,APO_FAC 50.0}
DECL E6POS XP306={x -92.6007004,y 2685.50098,z 861.002319,a 47.788929,b -0.179067105,c -89.6297226,s 6,t 51,e1 0.0,e2 0.0,e3 0.0,e4 0.0,e5 0.0,e6 0.0}
DECL FDAT Fp306={TOOL_NO 3,BASE_NO 0,IPO_FRAME #BASE}
DECL LDAT LCPDAT16={VEL 2.0,ACC 100.0,APO_DIST 100.0,APO_FAC 50.0}
DECL E6POS XP307={x -215.8311,y 2796.93311,z 760.875671,a 47.960289,b 0.0413109697,c -90.3944168,s 6,t 51,e1 0.0,e2 0.0,e3 0.0,e4 0.0,e5 0.0,e6 0.0}
DECL FDAT Fp307={TOOL_NO 3,BASE_NO 0,IPO_FRAME #BASE}
DECL LDAT LCPDAT17={VEL 2.0,ACC 100.0,APO_DIST 100.0,APO_FAC 50.0}
DECL E6POS XP308={x -249.264603,y 2416.05396,z 831.613281,a -13.6855202,b 56.5440903,c -155.689804,s 6,t 51,e1 0.0,e2 0.0,e3 0.0,e4 0.0,e5 0.0,e6 0.0}
DECL FDAT Fp308={TOOL_NO 8,BASE_NO 0,IPO_FRAME #BASE}
DECL LDAT LCPDAT18={VEL 2.0,ACC 100.0,APO_DIST 100.0,APO_FAC 50.0}
DECL PDAT PPDAT48={VEL 100.0,ACC 100.0,APO_DIST 100.0}
DECL E6POS XP2000={x 14.7387199,y 2430.83203,z 1561.30005,a 44.1596794,b -0.293628901,c -80.8446121,s 6,t 51,e1 0.0,e2 0.0,e3 0.0,e4 0.0,e5 0.0,e6 0.0}
DECL FDAT Fp2000={TOOL_NO 3,BASE_NO 0,IPO_FRAME #BASE}
DECL PDAT PPDAT49={VEL 100.0,ACC 100.0,APO_DIST 100.0}
DECL E6POS XP2001={x -207.498093,y 2790.38208,z 871.288025,a 47.096241,b 0.0432586595,c -89.4638367,s 6,t 51,e1 0.0,e2 0.0,e3 0.0,e4 0.0,e5 0.0,e6 0.0}
DECL FDAT Fp2001={TOOL_NO 3,BASE_NO 0,IPO_FRAME #BASE}
DECL PDAT PPDAT50={VEL 100.0,ACC 100.0,APO_DIST 100.0}
DECL E6POS XP2002={x -28.5181293,y 2384.37012,z 1449.54504,a 37.3302917,b 0.506031811,c -84.0773773,s 6,t 51,e1 0.0,e2 0.0,e3 0.0,e4 0.0,e5 0.0,e6 0.0}
DECL FDAT Fp2002={TOOL_NO 3,BASE_NO 0,IPO_FRAME #BASE}
DECL PDAT PPDAT51={VEL 100.0,ACC 100.0,APO_DIST 100.0}
DECL E6POS XP2003={x -109.917603,y 0.0234237108,z 210.146301,a 120.136902,b 15.4005804,c 90.5666122,s 2,t 2,e1 0.0,e2 0.0,e3 0.0,e4 0.0,e5 0.0,e6 0.0}
DECL FDAT Fp2003={TOOL_NO 8,BASE_NO 2,IPO_FRAME #BASE}
DECL PDAT PPDAT52={VEL 100.0,ACC 100.0,APO_DIST 100.0}
DECL E6POS XP2004={x -111.688004,y -0.708715677,z 218.358505,a 120.208,b 15.4733295,c 90.2876587,s 2,t 2,e1 0.0,e2 0.0,e3 0.0,e4 0.0,e5 0.0,e6 0.0}
DECL FDAT Fp2004={TOOL_NO 8,BASE_NO 2,IPO_FRAME #BASE}
DECL PDAT PPDAT53={VEL 100.0,ACC 100.0,APO_DIST 100.0}
DECL E6POS XP2005={x 2102.97998,y -1433.78003,z 797.644897,a 29.9009609,b 14.9999199,c 89.9971924,s 2,t 2,e1 0.0,e2 0.0,e3 0.0,e4 0.0,e5 0.0,e6 0.0}
DECL FDAT Fp2005={TOOL_NO 8,BASE_NO 0,IPO_FRAME #BASE}
DECL PDAT PPDAT54={VEL 100.0,ACC 100.0,APO_DIST 100.0}
DECL E6POS XPCORRECAO={x 3.59345198,y 1.01353002,z -95.5222626,a -112.648697,b 89.3137512,c -112.632202,s 2,t 2,e1 0.0,e2 0.0,e3 0.0,e4 0.0,e5 0.0,e6 0.0}
DECL FDAT FpCorrecao={TOOL_NO 3,BASE_NO 2,IPO_FRAME #BASE}
DECL LDAT LCPDAT19={VEL 2.0,ACC 100.0,APO_DIST 100.0,APO_FAC 50.0}
DECL PDAT PPDAT55={VEL 100.0,ACC 100.0,APO_DIST 100.0}
DECL PDAT PPDAT56={VEL 100.0,ACC 100.0,APO_DIST 100.0}
DECL E6POS XIII={x -504.836914,y -1.29663301,z -86.6123962,a -90.1386566,b 89.4559326,c -90.2674332,s 2,t 2,e1 0.0,e2 0.0,e3 0.0,e4 0.0,e5 0.0,e6 0.0}
DECL FDAT Fiii={TOOL_NO 3,BASE_NO 2,IPO_FRAME #BASE}
DECL E6POS XP1000={x 2102.33008,y -1536.07996,z 496.279785,a 43.0725784,b 89.5379486,c 133.203598,s 2,t 2,e1 0.0,e2 0.0,e3 0.0,e4 0.0,e5 0.0,e6 0.0}
DECL FDAT FP1000={TOOL_NO 3,BASE_NO 0,IPO_FRAME #BASE}
DECL LDAT LCPDAT20={VEL 2.0,ACC 85.0,APO_DIST 5.0,APO_FAC 50.0}
DECL E6POS XP1001={x 2030.31799,y -1316.20203,z 795.768921,a 29.8997993,b 14.6134596,c 89.9970398,s 2,t 2,e1 0.0,e2 0.0,e3 0.0,e4 0.0,e5 0.0,e6 0.0}
DECL FDAT FP1001={TOOL_NO 8,BASE_NO 0,IPO_FRAME #BASE}
DECL LDAT LCPDAT21={VEL 2.0,ACC 90.0,APO_DIST 20.0,APO_FAC 50.0}
DECL GRP_TYP GGDAT7={G_APO #NO,TIME 0.200000003,CTRL #OFF,DLY 0,DST 1}
DECL GRP_TYP GGDAT8={G_APO #NO,TIME 0.400000006,CTRL #OFF,DLY 0,DST 1}
DECL E6POS XP1110={x 1000.30798,y 1289.79797,z 2072.68408,a -39.348381,b -9.88963509,c -108.188698,s 2,t 3,e1 0.0,e2 0.0,e3 0.0,e4 0.0,e5 0.0,e6 0.0}
DECL FDAT Fp1110={TOOL_NO 3,BASE_NO 2,IPO_FRAME #BASE}
DECL PDAT PPDAT57={VEL 100.0,ACC 70.0,APO_DIST 10.0}
DECL E6AXIS Xp555={a1 19.1500206,a2 -32.0110703,a3 70.3853226,a4 125.674896,a5 53.9210014,a6 144.690994,e1 0.0,e2 0.0,e3 0.0,e4 0.0,e5 0.0,e6 0.0}
DECL FDAT Fp555={TOOL_NO 3,BASE_NO 2,IPO_FRAME #BASE}
DECL E6POS XP1111={x -2945.39404,y -1725.297,z 1956.93298,a -122.281799,b -45.4628716,c 124.668098,s 2,t 3,e1 0.0,e2 0.0,e3 0.0,e4 0.0,e5 0.0,e6 0.0}
DECL FDAT Fp1111={TOOL_NO 3,BASE_NO 2,IPO_FRAME #BASE}
DECL PDAT PPDAT58={VEL 100.0,ACC 70.0,APO_DIST 10.0}
DECL E6POS XPBF={x 2105.9751,y -1465.03894,z 498.409912,a 35.9188499,b 89.6157074,c 125.8367,s 2,t 2,e1 0.0,e2 0.0,e3 0.0,e4 0.0,e5 0.0,e6 0.0}
DECL FDAT Fpbf={TOOL_NO 3,BASE_NO 0,IPO_FRAME #BASE}
DECL LDAT LCPDAT24={VEL 2.0,ACC 80.0,APO_DIST 2.0,APO_FAC 50.0}
DECL PDAT PPDAT59={VEL 100.0,ACC 85.0,APO_DIST 10.0}
DECL E6POS XPOOOOO={x 4.70453119,y -2.03591394,z -86.1317825,a -106.403603,b 88.7964783,c -107.004997,s 2,t 2,e1 0.0,e2 0.0,e3 0.0,e4 0.0,e5 0.0,e6 0.0}
DECL FDAT Fpooooo={TOOL_NO 3,BASE_NO 2,IPO_FRAME #BASE}
DECL LDAT LCPDAT25={VEL 2.0,ACC 100.0,APO_DIST 100.0,APO_FAC 50.0}
DECL PDAT PPDAT60={VEL 100.0,ACC 100.0,APO_DIST 10.0}
DECL E6POS XPE5={x -272.044403,y -5.84646177,z -83.9034119,a -104.6343,b 88.8928223,c -105.115799,s 2,t 2,e1 0.0,e2 0.0,e3 0.0,e4 0.0,e5 0.0,e6 0.0}
DECL FDAT Fpe5={TOOL_NO 3,BASE_NO 2,IPO_FRAME #BASE}
DECL PDAT PPDAT61={VEL 100.0,ACC 80.0,APO_DIST 10.0}
DECL E6POS XPE6={x -1057.00696,y 600.567993,z 2451.78296,a 175.840103,b -72.5611572,c 179.209396,s 2,t 3,e1 0.0,e2 0.0,e3 0.0,e4 0.0,e5 0.0,e6 0.0}
DECL FDAT Fpe6={TOOL_NO 3,BASE_NO 0,IPO_FRAME #BASE}
DECL PDAT PPDAT62={VEL 100.0,ACC 100.0,APO_DIST 10.0}
DECL E6POS XPE7={x 361.5159,y 1414.83301,z 2512.08594,a 147.746506,b -44.78545,c 124.511803,s 2,t 3,e1 0.0,e2 0.0,e3 0.0,e4 0.0,e5 0.0,e6 0.0}
DECL FDAT Fpe7={TOOL_NO 3,BASE_NO 0,IPO_FRAME #BASE}
DECL PDAT PPDAT63={VEL 100.0,ACC 100.0,APO_DIST 30.0}
DECL E6POS XPE8={x 2238.80811,y -209.441406,z 551.882019,a 78.0304718,b 41.77882,c 151.181107,s 2,t 2,e1 0.0,e2 0.0,e3 0.0,e4 0.0,e5 0.0,e6 0.0}
DECL FDAT Fpe8={TOOL_NO 3,BASE_NO 0,IPO_FRAME #BASE}
DECL PDAT PPDAT64={VEL 100.0,ACC 100.0,APO_DIST 30.0}
DECL E6POS XPE9={x 2099.44189,y -1270.51196,z 502.9263,a 178.483704,b 89.5624619,c -91.9139862,s 2,t 2,e1 0.0,e2 0.0,e3 0.0,e4 0.0,e5 0.0,e6 0.0}
DECL FDAT Fpe9={TOOL_NO 3,BASE_NO 0,IPO_FRAME #BASE}
DECL PDAT PPDAT65={VEL 100.0,ACC 100.0,APO_DIST 10.0}
DECL E6POS XPE10={x 2168.69604,y -607.793579,z 520.700623,a 80.9914093,b 55.8017502,c 167.490005,s 2,t 2,e1 0.0,e2 0.0,e3 0.0,e4 0.0,e5 0.0,e6 0.0}
DECL FDAT Fpe10={TOOL_NO 3,BASE_NO 0,IPO_FRAME #BASE}
DECL PDAT PPDAT66={VEL 100.0,ACC 100.0,APO_DIST 10.0}
DECL E6POS XPE11={x 17.2454109,y 1.06276798,z -89.7810135,a -146.968094,b 89.4119034,c -147.1306,s 2,t 2,e1 0.0,e2 0.0,e3 0.0,e4 0.0,e5 0.0,e6 0.0}
DECL FDAT Fpe11={TOOL_NO 3,BASE_NO 2,IPO_FRAME #BASE}
DECL PDAT PPDAT67={VEL 100.0,ACC 100.0,APO_DIST 100.0}
DECL E6POS XPE12={x 2103.61401,y -1551.68604,z 491.369598,a 41.904541,b 89.8547592,c 132.6008,s 2,t 2,e1 0.0,e2 0.0,e3 0.0,e4 0.0,e5 0.0,e6 0.0}
DECL FDAT Fpe12={TOOL_NO 3,BASE_NO 0,IPO_FRAME #BASE}
DECL PDAT PPDAT68={VEL 100.0,ACC 85.0,APO_DIST 5.0}
DECL E6POS XPE13={x 2275.20093,y -436.23819,z 669.757202,a 35.523201,b 48.9097099,c 121.533203,s 2,t 2,e1 0.0,e2 0.0,e3 0.0,e4 0.0,e5 0.0,e6 0.0}
DECL FDAT Fpe13={TOOL_NO 3,BASE_NO 0,IPO_FRAME #BASE}
DECL PDAT PPDAT69={VEL 100.0,ACC 100.0,APO_DIST 100.0}
DECL E6POS XPE14={x 61.3286514,y 1354.46399,z 1483.37097,a -32.1679802,b 49.4948006,c -122.354202,s 2,t 35,e1 0.0,e2 0.0,e3 0.0,e4 0.0,e5 0.0,e6 0.0}
DECL FDAT Fpe14={TOOL_NO 8,BASE_NO 0,IPO_FRAME #BASE}
DECL PDAT PPDAT70={VEL 100.0,ACC 100.0,APO_DIST 100.0}
DECL E6POS XPE15={x 1113.87598,y 620.051392,z 1404.91394,a 66.4364624,b -66.97155,c 107.328201,s 2,t 3,e1 0.0,e2 0.0,e3 0.0,e4 0.0,e5 0.0,e6 0.0}
DECL FDAT Fpe15={TOOL_NO 8,BASE_NO 0,IPO_FRAME #BASE}
DECL PDAT PPDAT71={VEL 100.0,ACC 100.0,APO_DIST 100.0}
DECL E6POS XPE16={x 2104.48389,y -1551.28003,z 500.023712,a -76.8818512,b 89.2413177,c 13.0448599,s 2,t 2,e1 0.0,e2 0.0,e3 0.0,e4 0.0,e5 0.0,e6 0.0}
DECL FDAT Fpe16={TOOL_NO 3,BASE_NO 0,IPO_FRAME #BASE}
DECL LDAT LCPDAT26={VEL 2.0,ACC 85.0,APO_DIST 5.0,APO_FAC 50.0}
DECL E6POS XPE17={x 2102.3269,y -1516.76001,z 496.281586,a 43.1311493,b 89.5387268,c 133.2621,s 2,t 2,e1 0.0,e2 0.0,e3 0.0,e4 0.0,e5 0.0,e6 0.0}
DECL FDAT Fpe17={TOOL_NO 3,BASE_NO 0,IPO_FRAME #BASE}
DECL LDAT LCPDAT27={VEL 2.0,ACC 85.0,APO_DIST 100.0,APO_FAC 50.0}
DECL E6POS XPE18={x 2073.55005,y -1377.06494,z 791.333618,a 29.7421494,b 14.6915703,c 89.9213562,s 2,t 2,e1 0.0,e2 0.0,e3 0.0,e4 0.0,e5 0.0,e6 0.0}
DECL FDAT Fpe18={TOOL_NO 8,BASE_NO 0,IPO_FRAME #BASE}
DECL PDAT PPDAT72={VEL 100.0,ACC 100.0,APO_DIST 10.0}
DECL E6POS XPE19={x 2073.55005,y -1377.06494,z 791.330017,a 29.7420292,b 14.6916304,c 89.9213333,s 2,t 2,e1 0.0,e2 0.0,e3 0.0,e4 0.0,e5 0.0,e6 0.0}
DECL FDAT Fpe19={TOOL_NO 8,BASE_NO 0,IPO_FRAME #BASE}
DECL PDAT PPDAT73={VEL 100.0,ACC 100.0,APO_DIST 10.0}
DECL E6POS XPE20={x 2089.03809,y -1401.85596,z 795.66333,a 29.3717995,b 14.6907701,c 89.8277283,s 2,t 2,e1 0.0,e2 0.0,e3 0.0,e4 0.0,e5 0.0,e6 0.0}
DECL FDAT Fpe20={TOOL_NO 8,BASE_NO 0,IPO_FRAME #BASE}
DECL PDAT PPDAT74={VEL 100.0,ACC 100.0,APO_DIST 10.0}
DECL E6POS XPE21={x 2098.87695,y -1429.84399,z 801.184875,a 29.6556606,b 14.70996,c 90.0613937,s 2,t 2,e1 0.0,e2 0.0,e3 0.0,e4 0.0,e5 0.0,e6 0.0}
DECL FDAT Fpe21={TOOL_NO 8,BASE_NO 0,IPO_FRAME #BASE}
DECL LDAT LCPDAT28={VEL 2.0,ACC 80.0,APO_DIST 100.0,APO_FAC 50.0}
DECL LDAT LCPDAT29={VEL 2.0,ACC 80.0,APO_DIST 100.0,APO_FAC 50.0}
DECL LDAT LCPDAT30={VEL 2.0,ACC 80.0,APO_DIST 100.0,APO_FAC 50.0}
DECL E6POS XPE22={x 2248.53589,y -482.593689,z 618.861023,a 43.96315,b 53.1729584,c 132.135895,s 2,t 2,e1 0.0,e2 0.0,e3 0.0,e4 0.0,e5 0.0,e6 0.0}
DECL FDAT Fpe22={TOOL_NO 3,BASE_NO 0,IPO_FRAME #BASE}
DECL PDAT PPDAT75={VEL 100.0,ACC 100.0,APO_DIST 10.0}
DECL E6POS XPE23={x 2275.19507,y -436.238708,z 669.743713,a 35.5233803,b 48.9102211,c 121.533501,s 2,t 2,e1 0.0,e2 0.0,e3 0.0,e4 0.0,e5 0.0,e6 0.0}
DECL FDAT Fpe23={TOOL_NO 3,BASE_NO 0,IPO_FRAME #BASE}
DECL PDAT PPDAT76={VEL 100.0,ACC 100.0,APO_DIST 10.0}
DECL E6POS XPE24={x 2238.80811,y -209.438599,z 551.884888,a 78.0306625,b 41.7785301,c 151.181198,s 2,t 2,e1 0.0,e2 0.0,e3 0.0,e4 0.0,e5 0.0,e6 0.0}
DECL FDAT Fpe24={TOOL_NO 3,BASE_NO 0,IPO_FRAME #BASE}
DECL PDAT PPDAT77={VEL 100.0,ACC 100.0,APO_DIST 10.0}
ENDDAT
